Staubli VAL3: MsgRecvState.pjx

--- MsgRecvState.pjx ---
Parameters version=s7.8.1 stackSize=5000 millimeterUnit=true
Program file=start.pgx
Program file=stop.pgx
Data file=MsgRecvState.dtx

--- MsgRecvState.dtx ---
public num RECEIVE_HEADER
public num DECODE_HEADER
public num RECEIVE_BODY
public num DECODE_BODY
public num PUSH_MOTION
public num HANDLE_REQUEST
public num SEND_ACK
